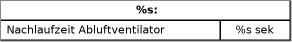
VISUALIZATION V_WCRaum  // 292x42
VAR_INPUT
	IN_Title		: STRING;
END_VAR
VAR_IN_OUT
	IO_fbWCRaum : FB_WCRaum;
END_VAR
    Rectangle (220,20 70x20), "%s sek", tooltip "Nach Abschalten des Bewegungsmelders läuft der Abluftventilator die hier eingestellte Zeit nach", text variable: IO_fbWCRaum.VdiAbluftNachlaufzeit
        OnMouseClick: write the text variable via Default, min 3, max 2000
    Rectangle (0,20 220x20), "Nachlaufzeit Abluftventilator", tooltip "Nach Abschalten des Bewegungsmelders läuft der Abluftventilator die hier eingestellte Zeit nach"
    Rectangle (0,0 290x20), "%s:", tooltip "Nach Abschalten des Bewegungsmelders läuft der Abluftventilator die hier eingestellte Zeit nach", text variable: IN_Title
END_VISUALIZATION

(* stored: Version 1.1.0.1, ProductVersion 3.1.4018.10
   Visu V_WCRaum: Id {a5e33bf6-8bfe-469f-abba-979aef687749} *)
